(* CODESYS project ControlAlgorithm.library
   Author: m.kleven@beckhoff.com
   Version: 0.0.2
   Description: Control Algorithms
   Title: ControlAlgorithm
   Placeholder: ControlAlgorithm
   Company: Beckhoff Automation LLC.

Project tree, tasks and I/O mapping:
  libraries: Tc2_System, * (Beckhoff Automation GmbH)
  Project Information/
    function F_GetCompany [ST]
    function F_GetTitle [ST]
    function F_GetVersion [ST]
  Version/
    global variables Global_Version
  data type E_FilterType
  function block FB_LowPassHighPassFilter [ST]
  function block FB_MovingAverage [ST]
  function block FB_PIDController [ST]
*)

// E_FilterType
{attribute 'qualified_only'}
{attribute 'strict'}
{attribute 'to_string'}
TYPE E_FilterType  :
(
   LowPass := 0,     // Low-pass filter
    HighPass := 1     // High-pass filter
);
END_TYPE

// Version/Global_Version
{attribute 'TcGenerated'}
{attribute 'no-analysis'}
{attribute 'linkalways'}
// This function has been automatically generated from the project information.
VAR_GLOBAL CONSTANT
	{attribute 'const_non_replaced'}
	stLibVersion_ControlAlgorithm : ST_LibVersion := (iMajor := 0, iMinor := 0, iBuild := 2, iRevision := 0, nFlags := 0, sVersion := '0.0.2');
END_VAR

// Project Information/F_GetCompany
// This function has been automatically generated from the project information.
{attribute 'signature_flag' := '1073741824'}
{attribute 'TcGenerated'}
{attribute 'no-analysis'}
FUNCTION F_GetCompany : WSTRING
VAR_INPUT
	
END_VAR

F_GetCompany := "Beckhoff Automation LLC.";

END_FUNCTION

// Project Information/F_GetTitle
// This function has been automatically generated from the project information.
{attribute 'signature_flag' := '1073741824'}
{attribute 'TcGenerated'}
{attribute 'no-analysis'}
FUNCTION F_GetTitle : WSTRING
VAR_INPUT
	
END_VAR

F_GetTitle := "ControlAlgorithm";

END_FUNCTION

// Project Information/F_GetVersion
// This function has been automatically generated from the project information.
{attribute 'signature_flag' := '1073741824'}
{attribute 'TcGenerated'}
{attribute 'no-analysis'}
FUNCTION F_GetVersion : ST_LibVersion
VAR_INPUT
	
END_VAR

F_GetVersion.iMajor := 0;
F_GetVersion.iMinor := 0;
F_GetVersion.iBuild := 2;
F_GetVersion.iRevision := 0;
F_GetVersion.sVersion := '0.0.2';
F_GetVersion.nFlags := 0;

END_FUNCTION

// FB_LowPassHighPassFilter
FUNCTION_BLOCK FB_LowPassHighPassFilter
VAR_INPUT
    Enable       : BOOL;                                // Enable filter
    Input        : LREAL;                               // Input signal
    FilterType   : E_FilterType := E_FilterType.LowPass; // Filter type selection
    CutoffFreq   : LREAL := 1.0;                       // Cutoff frequency in Hz
    Reset        : BOOL;                                // Reset filter state
END_VAR

VAR_OUTPUT
    Output       : LREAL;                               // Filtered output
    Error        : BOOL;                                // Error flag
END_VAR

VAR
    OutputPrevious : LREAL := 0.0;                      // Previous output value
    InputPrevious  : LREAL := 0.0;                      // Previous input value (for high-pass)
    Alpha          : LREAL;                             // Filter coefficient
    CycleTime      : LREAL := 0.001;                    // Cycle time in seconds
    TaskIdx        : DINT;
    FirstScan      : BOOL := TRUE;
END_VAR

IF FirstScan THEN
    FirstScan := FALSE;
    TaskIdx := GETCURTASKINDEXEX();
    IF TaskIdx > 0 THEN
        // Convert from 100ns units to seconds
        CycleTime := TO_LREAL(TwinCAT_SystemInfoVarList._TaskInfo[TaskIdx].CycleTime) / 10000000.0;
    END_IF
END_IF

IF Enable THEN
    // Input validation
    IF CutoffFreq <= 0.0 OR CycleTime <= 0.0 THEN
        Error := TRUE;
        Output := Input;  // Pass through on error
        RETURN;
    END_IF
    
    // Reset filter if requested
    IF Reset THEN
        OutputPrevious := Input;
        InputPrevious := Input;
    END_IF
    
    // Calculate filter coefficient (alpha)
    // For first-order filter: alpha = dt / (RC + dt)
    // Where RC = 1 / (2 * pi * fc), fc = cutoff frequency
    Alpha := CycleTime / ((1.0 / (2.0 * Tc2_System.PI * CutoffFreq)) + CycleTime);
    
    // Limit alpha to prevent numerical issues
    IF Alpha > 1.0 THEN
        Alpha := 1.0;
    ELSIF Alpha < 0.0 THEN
        Alpha := 0.0;
    END_IF
    
    // Apply appropriate filter
    CASE FilterType OF
        E_FilterType.LowPass:
            // Low-pass filter: y[n] = α * x[n] + (1-α) * y[n-1]
            Output := Alpha * Input + (1.0 - Alpha) * OutputPrevious;
            
        E_FilterType.HighPass:
            // High-pass filter: y[n] = α * (y[n-1] + x[n] - x[n-1])
            Output := Alpha * (OutputPrevious + Input - InputPrevious);
            
        ELSE
            Error := TRUE;
            Output := Input;
            RETURN;
    END_CASE
    
    // Store values for next iteration
    OutputPrevious := Output;
    InputPrevious := Input;
    Error := FALSE;
    
ELSE
    // Filter disabled - pass through input
    Output := Input;
    OutputPrevious := Input;
    InputPrevious := Input;
    Error := FALSE;
END_IF

END_FUNCTION_BLOCK

// FB_MovingAverage
FUNCTION_BLOCK FB_MovingAverage
VAR_INPUT
    Enable      : BOOL;           // Enable filter
    Input       : LREAL;          // Input signal to filter
    SampleCount : UDINT := 10;    // Number of samples in moving average (1-100)
    Reset       : BOOL;           // Reset filter buffer
END_VAR

VAR_OUTPUT
    Output      : LREAL;          // Filtered output
    Valid       : BOOL;           // Output is valid (buffer is full)
    Error       : BOOL;           // Error flag
END_VAR

VAR
    SampleBuffer : ARRAY[1..100] OF LREAL;  // Circular buffer for samples
    BufferIndex  : UDINT := 1;              // Current buffer index
    BufferSum    : LREAL := 0.0;            // Sum of all samples in buffer
    BufferFull   : BOOL := FALSE;           // Buffer has been filled once
    SamplesFilled : UDINT := 0;             // Number of valid samples in buffer
    LastSampleCount : UDINT := 0;           // Previous sample count for validation
END_VAR

VAR CONSTANT
    MaxSamples : UDINT := 100;    // Maximum number of samples
END_VAR

// Function block code
IF Enable THEN
    // Input validation
    IF SampleCount < 1 OR SampleCount > MaxSamples THEN
        Error := TRUE;
        Output := Input;  // Pass through on error
        Valid := FALSE;
        RETURN;
    END_IF
    
    // Reset buffer if requested or sample count changed
    IF Reset OR (SampleCount <> LastSampleCount) THEN
        // Clear the buffer
        FOR BufferIndex := 1 TO MaxSamples DO
            SampleBuffer[BufferIndex] := 0.0;
        END_FOR
        BufferIndex := 1;
        BufferSum := 0.0;
        BufferFull := FALSE;
        SamplesFilled := 0;
        LastSampleCount := SampleCount;
    END_IF
    
    // Remove old sample from sum if buffer position was previously used
    IF SamplesFilled >= SampleCount THEN
        BufferSum := BufferSum - SampleBuffer[BufferIndex];
    END_IF
    
    // Add new sample to buffer and sum
    SampleBuffer[BufferIndex] := Input;
    BufferSum := BufferSum + Input;
    
    // Update sample count
    IF SamplesFilled < SampleCount THEN
        SamplesFilled := SamplesFilled + 1;
    END_IF
    
    // Calculate moving average
    Output := BufferSum / TO_LREAL(SamplesFilled);
    
    // Update buffer index (circular buffer)
    BufferIndex := BufferIndex + 1;
    IF BufferIndex > SampleCount THEN
        BufferIndex := 1;
        BufferFull := TRUE;
    END_IF
    
    // Output is valid when we have enough samples
    Valid := (SamplesFilled >= SampleCount);
    Error := FALSE;
    
ELSE
    // Filter disabled - pass through input
    Output := Input;
    Valid := FALSE;
    Error := FALSE;
    
    // Reset buffer when disabled
    FOR BufferIndex := 1 TO MaxSamples DO
        SampleBuffer[BufferIndex] := 0.0;
    END_FOR
    BufferIndex := 1;
    BufferSum := 0.0;
    BufferFull := FALSE;
    SamplesFilled := 0;
END_IF

END_FUNCTION_BLOCK

// FB_PIDController
FUNCTION_BLOCK FB_PIDController
VAR_INPUT
	Enable		 : BOOL;		   // Enable PID controller
	Setpoint	 : LREAL;		   // Desired setpoint
	ProcessValue : LREAL;		   // Current process value (feedback)
	Kp			 : LREAL := 1.0;   // Proportional gain
	Ki			 : LREAL := 0.0;   // Integral gain
	Kd			 : LREAL := 0.0;   // Derivative gain
	OutputMin	 : LREAL := 0.0;   // Minimum output limit
	OutputMax	 : LREAL := 100.0; // Maximum output limit
	Reset		 : BOOL;		   // Reset integral accumulator
	ManualMode	 : BOOL;		   // Manual mode enable
	ManualOutput : LREAL := 0.0;   // Manual mode output value
END_VAR

VAR_OUTPUT
	Output		   : LREAL; // PID controller output
	Error		   : LREAL; // Current error (SP - PV)
	IntegralTerm   : LREAL; // Integral term value
	DerivativeTerm : LREAL; // Derivative term value
	Saturated	   : BOOL;	// Output is saturated
	ErrorFlag	   : BOOL;	// Error condition
END_VAR

VAR
	ErrorPrevious : LREAL;			// Previous error for derivative calculation
	IntegralSum	  : LREAL;			// Integral accumulator
	CycleTime	  : LREAL := 0.001; // Cycle time in seconds
	TaskIdx		  : DINT;
	FirstScan	  : BOOL := TRUE;
	OutputRaw	  : LREAL; // Raw output before limiting
END_VAR

IF FirstScan THEN
	FirstScan := FALSE;
	TaskIdx	  := GETCURTASKINDEXEX();
	IF TaskIdx > 0 THEN
		// Convert from 100ns units to seconds
		CycleTime := TO_LREAL(TwinCAT_SystemInfoVarList._TaskInfo[TaskIdx].CycleTime) / 10000000.0;
	END_IF
END_IF

IF Enable THEN
	// Calculate current error
	Error := Setpoint - ProcessValue;

	// Reset integral if requested or if in manual mode
	IF Reset OR ManualMode THEN
		IntegralSum := 0.0;
	END_IF

	// Manual mode operation
	IF ManualMode THEN
		Output		   := ManualOutput;
		IntegralTerm   := 0.0;
		DerivativeTerm := 0.0;
		Saturated	   := FALSE;
		ErrorFlag	   := FALSE;
		ErrorPrevious  := Error;
		RETURN;
	END_IF

	// Input validation
	IF CycleTime <= 0.0 OR OutputMax <= OutputMin THEN
		ErrorFlag := TRUE;
		Output	  := 0.0;
		RETURN;
	END_IF

	// Calculate integral term with windup protection
	IF NOT Saturated THEN
		IntegralSum := IntegralSum + (Error * CycleTime);
	END_IF

	IntegralTerm := Ki * IntegralSum;

	// Calculate derivative term
	DerivativeTerm := Kd * (Error - ErrorPrevious) / CycleTime;

	// Calculate raw PID output
	OutputRaw := (Kp * Error) + IntegralTerm + DerivativeTerm;

	// Apply output limits
	IF OutputRaw > OutputMax THEN
		Output	  := OutputMax;
		Saturated := TRUE;
	ELSIF OutputRaw < OutputMin THEN
		Output	  := OutputMin;
		Saturated := TRUE;
	ELSE
		Output	  := OutputRaw;
		Saturated := FALSE;
	END_IF

	// Store error for next derivative calculation
	ErrorPrevious := Error;
	ErrorFlag	  := FALSE;
ELSE
	// Controller disabled
	Output		   := 0.0;
	Error		   := 0.0;
	IntegralTerm   := 0.0;
	DerivativeTerm := 0.0;
	IntegralSum	   := 0.0;
	ErrorPrevious  := 0.0;
	Saturated	   := FALSE;
	ErrorFlag	   := FALSE;
END_IF

END_FUNCTION_BLOCK
